TYPE InitializationStates :
(
	SHUTDOWN := 0,
	INITIALIZING := 1,
	INITIALIZING_FAILED := 2,
	INITIALIZED := 3,
	LOCKED := 4
);
END_TYPE

(* stored: Version 1.1.0.1, ProductVersion 3.1.4019.2
   DUT InitializationStates: Id {60b5e1a7-ed54-4b56-b487-1e9acea05be0} *)
